// Mitsubishi GX Works2 project: data resister with counter   PLC: FX1N/FX1NC

PROGRAM MAIN
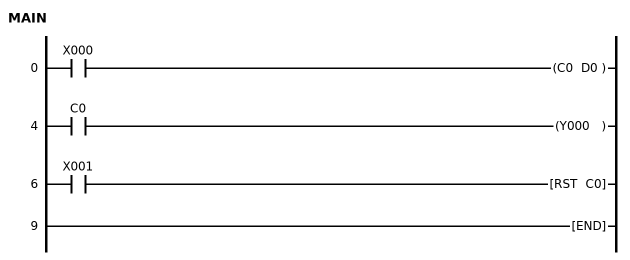
0     LD      X000
      OUT     C0 D0
4     LD      C0
      OUT     Y000
6     LD      X001
      RST     C0
9     END
END_PROGRAM
